//----------------------------------------------------------------------------//
//            Copyright 2018 Rieckermann Engineering Operations               //
//----------------------------------------------------------------------------//
// Description:                                                               //
// This file contains globally addressable event flags and data. The function //
// traverses the event datablock UDT structures to see if any event bits have //
// been raised. This is called each scan from the main program block OB1      //
// which therefore takes care of the looping required.                        //
//----------------------------------------------------------------------------//
// Revision history:                                                          //
// Rev By               Date        CC        Note                            //
// 2.0 David Paspa      16-May-2018 NA        Reboot design for S7-1500 not   //
//                                            using ALARM_D etc.              //
// 1.0 David Paspa      11-Apr-2018 NA        Initial design.                 //
//----------------------------------------------------------------------------//
FUNCTION_BLOCK "ifbEventLogReal"
TITLE = S7 Alarms for SFC log real data
{ S7_Optimized_Access := 'TRUE' }
AUTHOR : REO
NAME : ifbEventLogReal
VERSION : 2.0

//----------------------------------------------------------------------------//
// Declare variables:                                                         //
//----------------------------------------------------------------------------//
@@TEMPLATE_BEGIN@@
VAR
@@ATTR_BEGIN|pEventLogRealNum@@
    eventLogReal : Array[1..@@IDXEVENTMAX@@] of "udtEventLogReal";   // SFC events for logging real data
@@ATTR_END|pEventLogRealNum@@
@@ATTR_BEGIN|pEventLogRealAll@@
    Program_Alarm_@@IDXEVENT@@ : Program_Alarm;
@@ATTR_END|pEventLogRealAll@@
@@ATTR_BEGIN|pEventLogRealAll@@
    Alarm@@IDXEVENT@@_ErrorBit1 : Bool;
    Alarm@@IDXEVENT@@_ErrorBit2 : Bool;
    Alarm@@IDXEVENT@@_StatusWord1 : Word;
    Alarm@@IDXEVENT@@_StatusWord2 : Word;
    Alarm@@IDXEVENT@@_StateByte : Byte;
@@ATTR_END|pEventLogRealAll@@
	SourceData : Word;
END_VAR

VAR_TEMP
    almError : Bool;
    almState : Byte;
    almStatus : Word;
END_VAR

BEGIN
@@ATTR_BEGIN|pEventLogRealAll@@
NETWORK
TITLE = Raise message event if required
    //------------------------------------------------------------------------//
    // EVENT   EVENT   EVENT   EVENT   EVENT   EVENT   EVENT   EVENT   EVENT  //
    // EVENT   EVENT   EVENT   EVENT   EVENT   EVENT   EVENT   EVENT   EVENT  //
    //                                                                        //
    // Raise the log message event if requested. No acknowledge required:     //
    //------------------------------------------------------------------------//
    L @@IDXEVENT@@;
    T #SourceData;

    CALL #Program_Alarm_@@IDXEVENT@@
    (   SIG       := #eventLogReal[@@IDXEVENT@@].trigger ,
		SD_1      := #SourceData ,
		SD_2      := #eventLogReal[@@IDXEVENT@@].dataValue ,
        Error     := #Alarm@@IDXEVENT@@_ErrorBit1 ,
        Status    := #Alarm@@IDXEVENT@@_StatusWord1
    );

@@ATTR_END|pEventLogRealAll@@

@@TEMPLATE_END@@
END_FUNCTION_BLOCK
